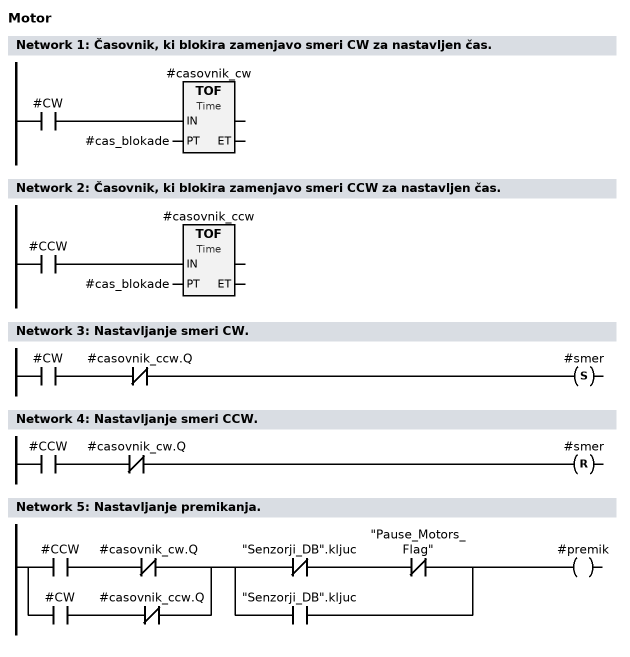
   #casovnik_cw.TOF(IN := #CW, PT := #cas_blokade);
END_REGION

REGION Network 2: Časovnik, ki blokira zamenjavo smeri CCW za nastavljen čas.
   #casovnik_ccw.TOF(IN := #CCW, PT := #cas_blokade);
END_REGION

REGION Network 3: Nastavljanje smeri CW.
   RUNG wire#powerrail
      Contact( #CW )
      I_Contact( #casovnik_ccw.Q )
      S_Coil( #smer )
   END_RUNG
   // the same network as SCL:
   IF #CW AND NOT #casovnik_ccw.Q THEN #smer := TRUE; END_IF;
END_REGION

REGION Network 4: Nastavljanje smeri CCW.
   RUNG wire#powerrail
      Contact( #CCW )
      I_Contact( #casovnik_cw.Q )
      R_Coil( #smer )
   END_RUNG
   // the same network as SCL:
   IF #CCW AND NOT #casovnik_cw.Q THEN #smer := FALSE; END_IF;
END_REGION

REGION Network 5: Nastavljanje premikanja.
   RUNG wire#powerrail
      Contact( #CCW )
      I_Contact( #casovnik_cw.Q )
      wire#w1
      I_Contact( "Senzorji_DB".kljuc )
      I_Contact( "Pause_Motors_Flag" )
      wire#w2
      Coil( #premik )
   END_RUNG
   RUNG wire#powerrail
      Contact( #CW )
      I_Contact( #casovnik_ccw.Q )
   END_RUNG wire#w1
   RUNG wire#w1
      Contact( "Senzorji_DB".kljuc )
   END_RUNG wire#w2
   // the same network as SCL:
   #premik := ((#CCW AND NOT #casovnik_cw.Q) OR (#CW AND NOT #casovnik_ccw.Q)) AND ((NOT "Senzorji_DB".kljuc AND NOT "Pause_Motors_Flag") OR "Senzorji_DB".kljuc);
END_REGION
END_FUNCTION_BLOCK

FUNCTION_BLOCK "Motorji"   // FB3, LAD
TITLE = Nastavljanje vseh različnih motorjev.
{ S7_Optimized_Access := 'FALSE' }
VERSION : 0.1
BEGIN

REGION Network 1: Izbira motorja
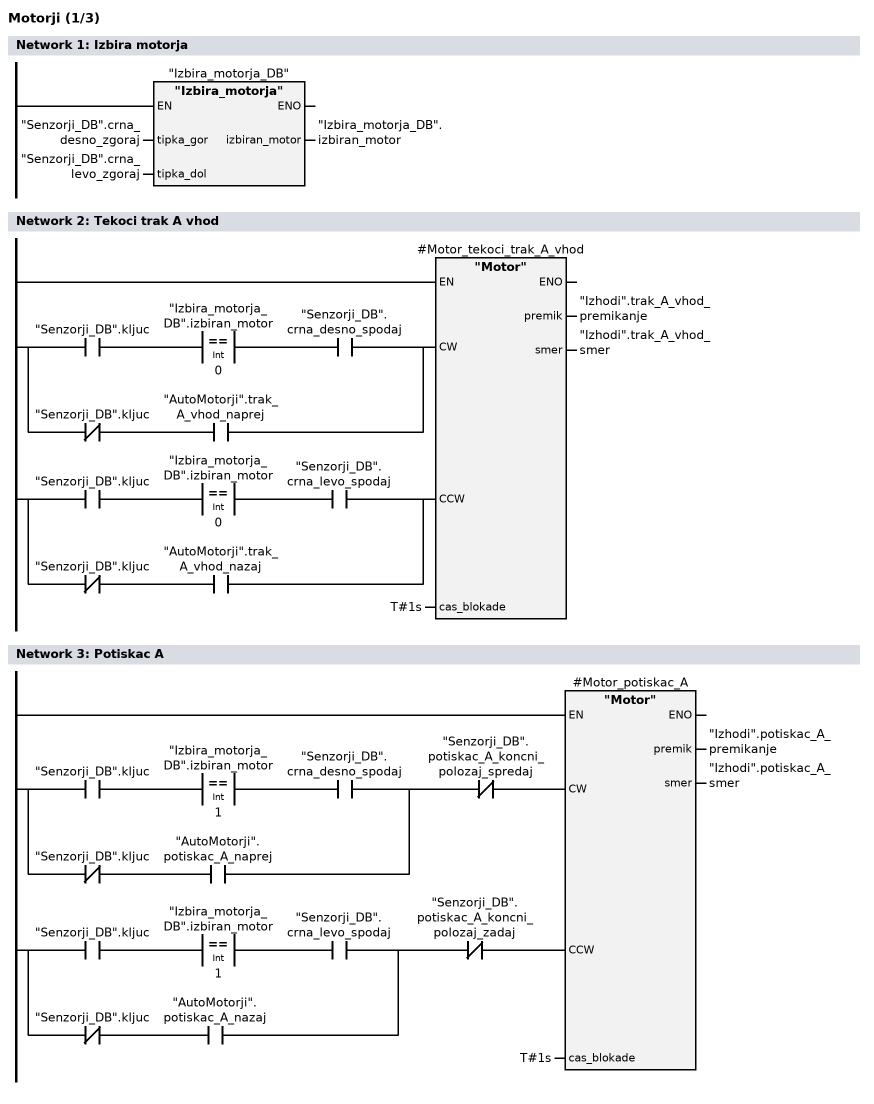
   RUNG wire#powerrail
      "Izbira_motorja_DB"(tipka_gor := "Senzorji_DB".crna_desno_zgoraj, tipka_dol := "Senzorji_DB".crna_levo_zgoraj, izbiran_motor => "Izbira_motorja_DB".izbiran_motor)
   END_RUNG
   // the same network as SCL:
   "Izbira_motorja_DB"(tipka_gor := "Senzorji_DB".crna_desno_zgoraj,   // "Izbira_motorja"
                       tipka_dol := "Senzorji_DB".crna_levo_zgoraj,
                       izbiran_motor => "Izbira_motorja_DB".izbiran_motor);
END_REGION

REGION Network 2: Tekoci trak A vhod
   RUNG wire#powerrail
      #Motor_tekoci_trak_A_vhod(CW := wire#w1, CCW := wire#w2, cas_blokade := T#1s, premik => "Izhodi".trak_A_vhod_premikanje, smer => "Izhodi".trak_A_vhod_smer)
   END_RUNG
   RUNG wire#powerrail
      Contact( "Senzorji_DB".kljuc )
      { S7_Templates := "SrcType := Int" } EQ_Contact(in1 := "Izbira_motorja_DB".izbiran_motor, in2 := 0)
      Contact( "Senzorji_DB".crna_desno_spodaj )
   END_RUNG wire#w1
   RUNG wire#powerrail
      I_Contact( "Senzorji_DB".kljuc )
      Contact( "AutoMotorji".trak_A_vhod_naprej )
   END_RUNG wire#w1
   RUNG wire#powerrail
      Contact( "Senzorji_DB".kljuc )
      { S7_Templates := "SrcType := Int" } EQ_Contact(in1 := "Izbira_motorja_DB".izbiran_motor, in2 := 0)
      Contact( "Senzorji_DB".crna_levo_spodaj )
   END_RUNG wire#w2
   RUNG wire#powerrail
      I_Contact( "Senzorji_DB".kljuc )
      Contact( "AutoMotorji".trak_A_vhod_nazaj )
   END_RUNG wire#w2
   // the same network as SCL:
   #Motor_tekoci_trak_A_vhod(CW := ("Senzorji_DB".kljuc AND ("Izbira_motorja_DB".izbiran_motor = 0) AND "Senzorji_DB".crna_desno_spodaj) OR (NOT "Senzorji_DB".kljuc AND "AutoMotorji".trak_A_vhod_naprej),   // "Motor"
                           CCW := ("Senzorji_DB".kljuc AND ("Izbira_motorja_DB".izbiran_motor = 0) AND "Senzorji_DB".crna_levo_spodaj) OR (NOT "Senzorji_DB".kljuc AND "AutoMotorji".trak_A_vhod_nazaj),
                           cas_blokade := T#1s,
                           premik => "Izhodi".trak_A_vhod_premikanje,
                           smer => "Izhodi".trak_A_vhod_smer);
END_REGION

REGION Network 3: Potiskac A
   RUNG wire#powerrail
      #Motor_potiskac_A(CW := wire#w2, CCW := wire#w4, cas_blokade := T#1s, premik => "Izhodi".potiskac_A_premikanje, smer => "Izhodi".potiskac_A_smer)
   END_RUNG
   RUNG wire#powerrail
      Contact( "Senzorji_DB".kljuc )
      { S7_Templates := "SrcType := Int" } EQ_Contact(in1 := "Izbira_motorja_DB".izbiran_motor, in2 := 1)
      Contact( "Senzorji_DB".crna_desno_spodaj )
      wire#w1
      I_Contact( "Senzorji_DB".potiskac_A_koncni_polozaj_spredaj )
   END_RUNG wire#w2
   RUNG wire#powerrail
      I_Contact( "Senzorji_DB".kljuc )
      Contact( "AutoMotorji".potiskac_A_naprej )
   END_RUNG wire#w1
   RUNG wire#powerrail
      Contact( "Senzorji_DB".kljuc )
      { S7_Templates := "SrcType := Int" } EQ_Contact(in1 := "Izbira_motorja_DB".izbiran_motor, in2 := 1)
      Contact( "Senzorji_DB".crna_levo_spodaj )
      wire#w3
      I_Contact( "Senzorji_DB".potiskac_A_koncni_polozaj_zadaj )
   END_RUNG wire#w4
   RUNG wire#powerrail
      I_Contact( "Senzorji_DB".kljuc )
      Contact( "AutoMotorji".potiskac_A_nazaj )
   END_RUNG wire#w3
   // the same network as SCL:
   #Motor_potiskac_A(CW := (("Senzorji_DB".kljuc AND ("Izbira_motorja_DB".izbiran_motor = 1) AND "Senzorji_DB".crna_desno_spodaj) OR (NOT "Senzorji_DB".kljuc AND "AutoMotorji".potiskac_A_naprej)) AND NOT "Senzorji_DB".potiskac_A_koncni_polozaj_spredaj,   // "Motor"
                     CCW := (("Senzorji_DB".kljuc AND ("Izbira_motorja_DB".izbiran_motor = 1) AND "Senzorji_DB".crna_levo_spodaj) OR (NOT "Senzorji_DB".kljuc AND "AutoMotorji".potiskac_A_nazaj)) AND NOT "Senzorji_DB".potiskac_A_koncni_polozaj_zadaj,
                     cas_blokade := T#1s,
                     premik => "Izhodi".potiskac_A_premikanje,
                     smer => "Izhodi".potiskac_A_smer);
END_REGION

REGION Network 4: Tekoci trak A stroj
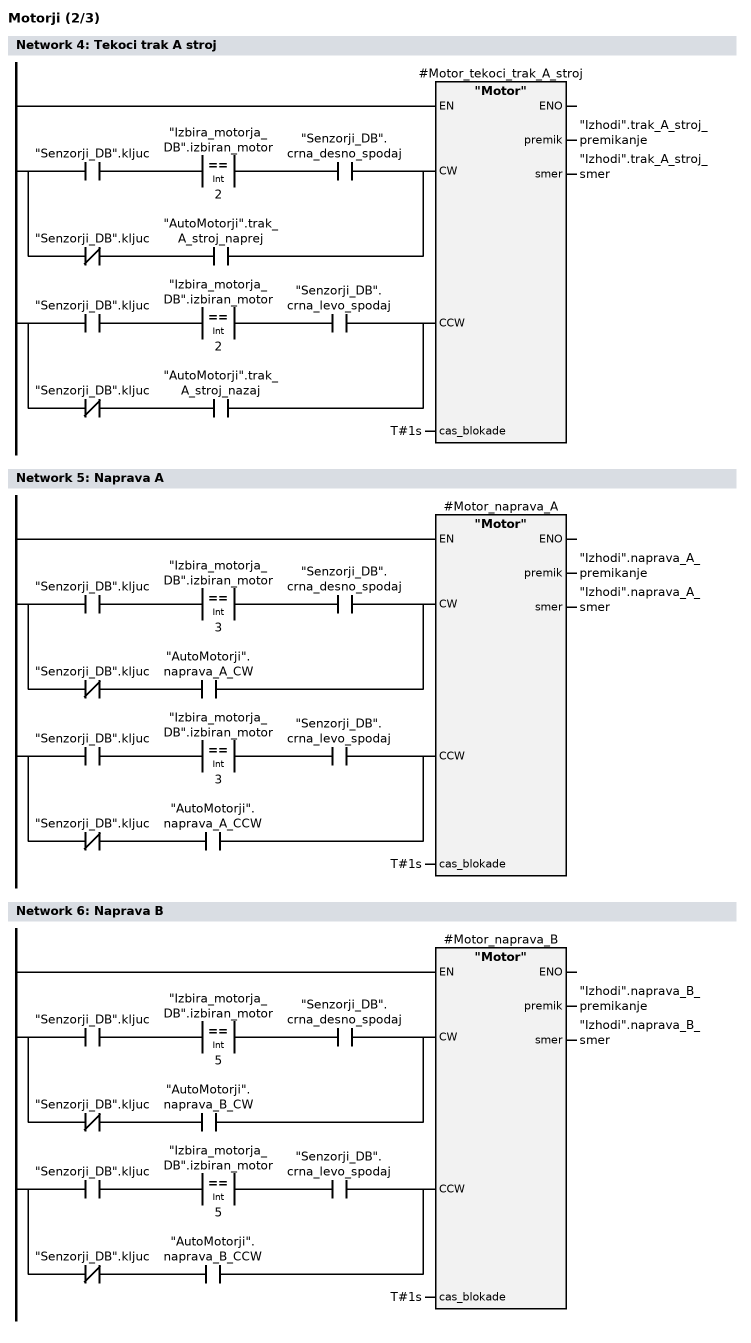
   RUNG wire#powerrail
      #Motor_tekoci_trak_A_stroj(CW := wire#w1, CCW := wire#w2, cas_blokade := T#1s, premik => "Izhodi".trak_A_stroj_premikanje, smer => "Izhodi".trak_A_stroj_smer)
   END_RUNG
   RUNG wire#powerrail
      Contact( "Senzorji_DB".kljuc )
      { S7_Templates := "SrcType := Int" } EQ_Contact(in1 := "Izbira_motorja_DB".izbiran_motor, in2 := 2)
      Contact( "Senzorji_DB".crna_desno_spodaj )
   END_RUNG wire#w1
   RUNG wire#powerrail
      I_Contact( "Senzorji_DB".kljuc )
      Contact( "AutoMotorji".trak_A_stroj_naprej )
   END_RUNG wire#w1
   RUNG wire#powerrail
      Contact( "Senzorji_DB".kljuc )
      { S7_Templates := "SrcType := Int" } EQ_Contact(in1 := "Izbira_motorja_DB".izbiran_motor, in2 := 2)
      Contact( "Senzorji_DB".crna_levo_spodaj )
   END_RUNG wire#w2
   RUNG wire#powerrail
      I_Contact( "Senzorji_DB".kljuc )
      Contact( "AutoMotorji".trak_A_stroj_nazaj )
   END_RUNG wire#w2
   // the same network as SCL:
   #Motor_tekoci_trak_A_stroj(CW := ("Senzorji_DB".kljuc AND ("Izbira_motorja_DB".izbiran_motor = 2) AND "Senzorji_DB".crna_desno_spodaj) OR (NOT "Senzorji_DB".kljuc AND "AutoMotorji".trak_A_stroj_naprej),   // "Motor"
                           CCW := ("Senzorji_DB".kljuc AND ("Izbira_motorja_DB".izbiran_motor = 2) AND "Senzorji_DB".crna_levo_spodaj) OR (NOT "Senzorji_DB".kljuc AND "AutoMotorji".trak_A_stroj_nazaj),
                           cas_blokade := T#1s,
                           premik => "Izhodi".trak_A_stroj_premikanje,
                           smer => "Izhodi".trak_A_stroj_smer);
END_REGION

REGION Network 5: Naprava A
   RUNG wire#powerrail
      #Motor_naprava_A(CW := wire#w1, CCW := wire#w2, cas_blokade := T#1s, premik => "Izhodi".naprava_A_premikanje, smer => "Izhodi".naprava_A_smer)
   END_RUNG
   RUNG wire#powerrail
      Contact( "Senzorji_DB".kljuc )
      { S7_Templates := "SrcType := Int" } EQ_Contact(in1 := "Izbira_motorja_DB".izbiran_motor, in2 := 3)
      Contact( "Senzorji_DB".crna_desno_spodaj )
   END_RUNG wire#w1
   RUNG wire#powerrail
      I_Contact( "Senzorji_DB".kljuc )
      Contact( "AutoMotorji".naprava_A_CW )
   END_RUNG wire#w1
   RUNG wire#powerrail
      Contact( "Senzorji_DB".kljuc )
      { S7_Templates := "SrcType := Int" } EQ_Contact(in1 := "Izbira_motorja_DB".izbiran_motor, in2 := 3)
      Contact( "Senzorji_DB".crna_levo_spodaj )
   END_RUNG wire#w2
   RUNG wire#powerrail
      I_Contact( "Senzorji_DB".kljuc )
      Contact( "AutoMotorji".naprava_A_CCW )
   END_RUNG wire#w2
   // the same network as SCL:
   #Motor_naprava_A(CW := ("Senzorji_DB".kljuc AND ("Izbira_motorja_DB".izbiran_motor = 3) AND "Senzorji_DB".crna_desno_spodaj) OR (NOT "Senzorji_DB".kljuc AND "AutoMotorji".naprava_A_CW),   // "Motor"
                    CCW := ("Senzorji_DB".kljuc AND ("Izbira_motorja_DB".izbiran_motor = 3) AND "Senzorji_DB".crna_levo_spodaj) OR (NOT "Senzorji_DB".kljuc AND "AutoMotorji".naprava_A_CCW),
                    cas_blokade := T#1s,
                    premik => "Izhodi".naprava_A_premikanje,
                    smer => "Izhodi".naprava_A_smer);
END_REGION

REGION Network 6: Naprava B
   RUNG wire#powerrail
      #Motor_naprava_B(CW := wire#w1, CCW := wire#w2, cas_blokade := T#1s, premik => "Izhodi".naprava_B_premikanje, smer => "Izhodi".naprava_B_smer)
   END_RUNG
   RUNG wire#powerrail
      Contact( "Senzorji_DB".kljuc )
      { S7_Templates := "SrcType := Int" } EQ_Contact(in1 := "Izbira_motorja_DB".izbiran_motor, in2 := 5)
      Contact( "Senzorji_DB".crna_desno_spodaj )
   END_RUNG wire#w1
   RUNG wire#powerrail
      I_Contact( "Senzorji_DB".kljuc )
      Contact( "AutoMotorji".naprava_B_CW )
   END_RUNG wire#w1
   RUNG wire#powerrail
      Contact( "Senzorji_DB".kljuc )
      { S7_Templates := "SrcType := Int" } EQ_Contact(in1 := "Izbira_motorja_DB".izbiran_motor, in2 := 5)
      Contact( "Senzorji_DB".crna_levo_spodaj )
   END_RUNG wire#w2
   RUNG wire#powerrail
      I_Contact( "Senzorji_DB".kljuc )
      Contact( "AutoMotorji".naprava_B_CCW )
   END_RUNG wire#w2
   // the same network as SCL:
   #Motor_naprava_B(CW := ("Senzorji_DB".kljuc AND ("Izbira_motorja_DB".izbiran_motor = 5) AND "Senzorji_DB".crna_desno_spodaj) OR (NOT "Senzorji_DB".kljuc AND "AutoMotorji".naprava_B_CW),   // "Motor"
                    CCW := ("Senzorji_DB".kljuc AND ("Izbira_motorja_DB".izbiran_motor = 5) AND "Senzorji_DB".crna_levo_spodaj) OR (NOT "Senzorji_DB".kljuc AND "AutoMotorji".naprava_B_CCW),
                    cas_blokade := T#1s,
                    premik => "Izhodi".naprava_B_premikanje,
                    smer => "Izhodi".naprava_B_smer);
END_REGION

REGION Network 7: Tekoci trak B stroj
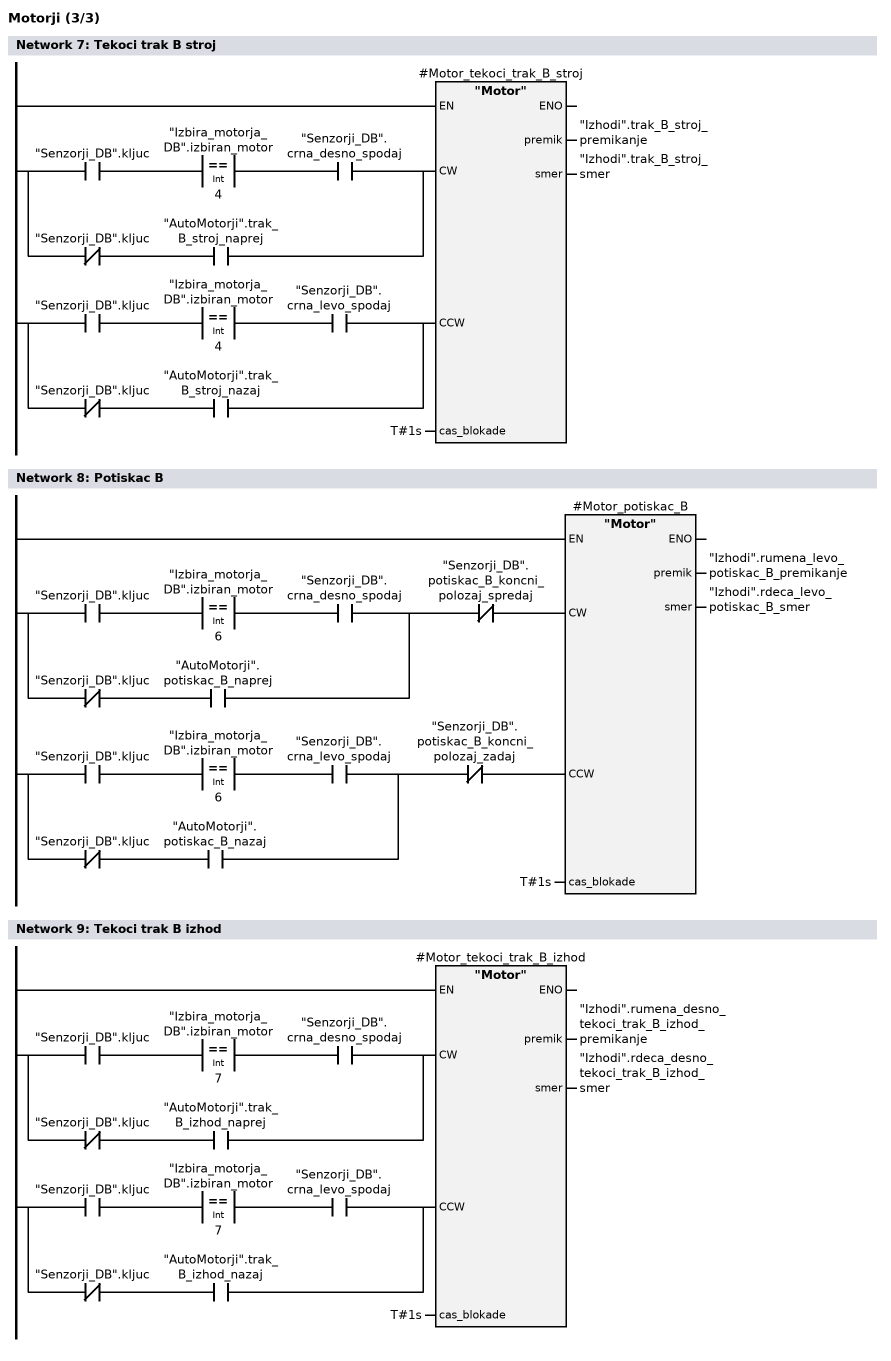
   RUNG wire#powerrail
      #Motor_tekoci_trak_B_stroj(CW := wire#w1, CCW := wire#w2, cas_blokade := T#1s, premik => "Izhodi".trak_B_stroj_premikanje, smer => "Izhodi".trak_B_stroj_smer)
   END_RUNG
   RUNG wire#powerrail
      Contact( "Senzorji_DB".kljuc )
      { S7_Templates := "SrcType := Int" } EQ_Contact(in1 := "Izbira_motorja_DB".izbiran_motor, in2 := 4)
      Contact( "Senzorji_DB".crna_desno_spodaj )
   END_RUNG wire#w1
   RUNG wire#powerrail
      I_Contact( "Senzorji_DB".kljuc )
      Contact( "AutoMotorji".trak_B_stroj_naprej )
   END_RUNG wire#w1
   RUNG wire#powerrail
      Contact( "Senzorji_DB".kljuc )
      { S7_Templates := "SrcType := Int" } EQ_Contact(in1 := "Izbira_motorja_DB".izbiran_motor, in2 := 4)
      Contact( "Senzorji_DB".crna_levo_spodaj )
   END_RUNG wire#w2
   RUNG wire#powerrail
      I_Contact( "Senzorji_DB".kljuc )
      Contact( "AutoMotorji".trak_B_stroj_nazaj )
   END_RUNG wire#w2
   // the same network as SCL:
   #Motor_tekoci_trak_B_stroj(CW := ("Senzorji_DB".kljuc AND ("Izbira_motorja_DB".izbiran_motor = 4) AND "Senzorji_DB".crna_desno_spodaj) OR (NOT "Senzorji_DB".kljuc AND "AutoMotorji".trak_B_stroj_naprej),   // "Motor"
                           CCW := ("Senzorji_DB".kljuc AND ("Izbira_motorja_DB".izbiran_motor = 4) AND "Senzorji_DB".crna_levo_spodaj) OR (NOT "Senzorji_DB".kljuc AND "AutoMotorji".trak_B_stroj_nazaj),
                           cas_blokade := T#1s,
                           premik => "Izhodi".trak_B_stroj_premikanje,
                           smer => "Izhodi".trak_B_stroj_smer);
END_REGION

REGION Network 8: Potiskac B
   RUNG wire#powerrail
      #Motor_potiskac_B(CW := wire#w2, CCW := wire#w4, cas_blokade := T#1s, premik => "Izhodi".rumena_levo_potiskac_B_premikanje, smer => "Izhodi".rdeca_levo_potiskac_B_smer)
   END_RUNG
   RUNG wire#powerrail
      Contact( "Senzorji_DB".kljuc )
      { S7_Templates := "SrcType := Int" } EQ_Contact(in1 := "Izbira_motorja_DB".izbiran_motor, in2 := 6)
      Contact( "Senzorji_DB".crna_desno_spodaj )
      wire#w1
      I_Contact( "Senzorji_DB".potiskac_B_koncni_polozaj_spredaj )
   END_RUNG wire#w2
   RUNG wire#powerrail
      I_Contact( "Senzorji_DB".kljuc )
      Contact( "AutoMotorji".potiskac_B_naprej )
   END_RUNG wire#w1
   RUNG wire#powerrail
      Contact( "Senzorji_DB".kljuc )
      { S7_Templates := "SrcType := Int" } EQ_Contact(in1 := "Izbira_motorja_DB".izbiran_motor, in2 := 6)
      Contact( "Senzorji_DB".crna_levo_spodaj )
      wire#w3
      I_Contact( "Senzorji_DB".potiskac_B_koncni_polozaj_zadaj )
   END_RUNG wire#w4
   RUNG wire#powerrail
      I_Contact( "Senzorji_DB".kljuc )
      Contact( "AutoMotorji".potiskac_B_nazaj )
   END_RUNG wire#w3
   // the same network as SCL:
   #Motor_potiskac_B(CW := (("Senzorji_DB".kljuc AND ("Izbira_motorja_DB".izbiran_motor = 6) AND "Senzorji_DB".crna_desno_spodaj) OR (NOT "Senzorji_DB".kljuc AND "AutoMotorji".potiskac_B_naprej)) AND NOT "Senzorji_DB".potiskac_B_koncni_polozaj_spredaj,   // "Motor"
                     CCW := (("Senzorji_DB".kljuc AND ("Izbira_motorja_DB".izbiran_motor = 6) AND "Senzorji_DB".crna_levo_spodaj) OR (NOT "Senzorji_DB".kljuc AND "AutoMotorji".potiskac_B_nazaj)) AND NOT "Senzorji_DB".potiskac_B_koncni_polozaj_zadaj,
                     cas_blokade := T#1s,
                     premik => "Izhodi".rumena_levo_potiskac_B_premikanje,
                     smer => "Izhodi".rdeca_levo_potiskac_B_smer);
END_REGION

REGION Network 9: Tekoci trak B izhod
   RUNG wire#powerrail
      #Motor_tekoci_trak_B_izhod(CW := wire#w1, CCW := wire#w2, cas_blokade := T#1s, premik => "Izhodi".rumena_desno_tekoci_trak_B_izhod_premikanje, smer => "Izhodi".rdeca_desno_tekoci_trak_B_izhod_smer)
   END_RUNG
   RUNG wire#powerrail
      Contact( "Senzorji_DB".kljuc )
      { S7_Templates := "SrcType := Int" } EQ_Contact(in1 := "Izbira_motorja_DB".izbiran_motor, in2 := 7)
      Contact( "Senzorji_DB".crna_desno_spodaj )
   END_RUNG wire#w1
   RUNG wire#powerrail
      I_Contact( "Senzorji_DB".kljuc )
      Contact( "AutoMotorji".trak_B_izhod_naprej )
   END_RUNG wire#w1
   RUNG wire#powerrail
      Contact( "Senzorji_DB".kljuc )
      { S7_Templates := "SrcType := Int" } EQ_Contact(in1 := "Izbira_motorja_DB".izbiran_motor, in2 := 7)
      Contact( "Senzorji_DB".crna_levo_spodaj )
   END_RUNG wire#w2
   RUNG wire#powerrail
      I_Contact( "Senzorji_DB".kljuc )
      Contact( "AutoMotorji".trak_B_izhod_nazaj )
   END_RUNG wire#w2
   // the same network as SCL:
   #Motor_tekoci_trak_B_izhod(CW := ("Senzorji_DB".kljuc AND ("Izbira_motorja_DB".izbiran_motor = 7) AND "Senzorji_DB".crna_desno_spodaj) OR (NOT "Senzorji_DB".kljuc AND "AutoMotorji".trak_B_izhod_naprej),   // "Motor"
                           CCW := ("Senzorji_DB".kljuc AND ("Izbira_motorja_DB".izbiran_motor = 7) AND "Senzorji_DB".crna_levo_spodaj) OR (NOT "Senzorji_DB".kljuc AND "AutoMotorji".trak_B_izhod_nazaj),
                           cas_blokade := T#1s,
                           premik => "Izhodi".rumena_desno_tekoci_trak_B_izhod_premikanje,
                           smer => "Izhodi".rdeca_desno_tekoci_trak_B_izhod_smer);
END_REGION
END_FUNCTION_BLOCK

(* ===== HMI "HMI_RT_1" =====
connection "HMI_Connection_1": ETHERNET, SIMATIC S7 300/400 MPI

HMI tags "Default tag table"
   "SCADA_alarm_aktive_globalno" : Bool, 100 ms
   "SCADA_alarm_potrditev" : Bool, 100 ms
   "SCADA_alarmi" : Word, 100 ms
   "SCADA_recept_vrtanje1" : Bool, 100 ms
   "SCADA_recept_cas_vrtanja1" : Time, 100 ms
   "SCADA_recept_vrtanje2" : Bool, 100 ms
   "SCADA_recept_cas_vrtanja2" : Time, 100 ms
   "SCADA_recept_smer_1" : Bool, 100 ms
   "SCADA_recept_smer_2" : Bool, 100 ms
   "Lokacije_DB_L1_vhod_1_zasedenost" : Bool, 100 ms
   "L1_L2_CNT_CV" : Int, 100 ms
   "Lokacije_DB_L2_vhod_2_zasedenost" : Bool, 100 ms
   "L2_L3_CNT_CV" : Int, 100 ms
   "Lokacije_DB_L3_potiskac_A_zasedenost" : Bool, 100 ms
   "L3_L4_CNT_CV" : Int, 100 ms
   "Lokacije_DB_L4_naprava_A_zasedenost" : Bool, 100 ms
   "Lokacije_DB_L5_naprava_B_zasedenost" : Bool, 100 ms
   "Lokacije_DB_L6_potiskac_B_zasedenost" : Bool, 100 ms
   "Lokacije_DB_L7_izhod_zasedenost" : Bool, 100 ms
   "SCADAVisual_DB_l3_l4_visibily" : Bool, 100 ms
   "L4_L5_CNT_CV" : Int, 100 ms
   "L5_L6_CNT_CV" : Int, 100 ms
   "L6_L7_CNT_CV" : Int, 100 ms
   "SCADAVisual_DB_l6_l7_visibily" : Bool, 100 ms
   "Senzorji_DB_fotocelica_material_na_vhodu" : Bool, 100 ms
   "Senzorji_DB_fotocelica_materal_pred_potiskacem" : Bool, 100 ms
   "Senzorji_DB_fotocelica_material_pod_napravo_A" : Bool, 100 ms
   "Senzorji_DB_fotocelica_material_pod_napravo_B" : Bool, 100 ms
   "Senzorji_DB_fotocelica_material_na_izhodu" : Bool, 100 ms
   "Senzorji_DB_potiskac_A_koncni_polozaj_zadaj" : Bool, 100 ms
   "Senzorji_DB_potiskac_A_koncni_polozaj_spredaj" : Bool, 100 ms
   "SCADAVisual_DB_potiskac_A_levo" : Bool, 100 ms
   "SCADAVisual_DB_potiskac_A_desno" : Bool, 100 ms
   "SCADAVisual_DB;potiskac_B_dol" : Bool, 100 ms
   "SCADAVisual_DB;potiskac_B_gor" : Bool, 100 ms
   "Senzorji_DB;potiskac_B_koncni_polozaj_zadaj" : Bool, 100 ms
   "Senzorji_DB;potiskac_B_koncni_polozaj_spredaj" : Bool, 100 ms
   "SCADAVisual_DB;trak_vhod_nazaj" : Bool, 100 ms
   "SCADAVisual_DB;trak_vhod_naprej" : Bool, 100 ms
   "SCADAVisual_DB;trak_A_naprej" : Bool, 100 ms
   "SCADAVisual_DB;trak_A_nazaj" : Bool, 100 ms
   "SCADAVisual_DB;trak_B_nazaj" : Bool, 100 ms
   "SCADAVisual_DB;trak_izhod_naprej" : Bool, 100 ms
   "SCADAVisual_DB;trak_izhod_nazaj" : Bool, 100 ms
   "SCADAVisual_DB;trak_B_naprej" : Bool, 100 ms
   "SCADAVisual_DB;l3_visibility" : Bool, 100 ms
   "SCADAVisual_DB;l6_visibility" : Bool, 100 ms
   "Auto_2_A_Naprava_DB;casVrtanja" : DInt, 100 ms
   "Auto_2_A_Naprava_DB;maxCasVrtanja" : DInt, 100 ms
   "Auto_3_B_Naprava_DB;casVrtanja" : DInt, 100 ms
   "Auto_3_B_Naprava_DB;maxCasVrtanja" : DInt, 100 ms
   "Lokacije_DB;L1_vhod_1;ID" : Int, 100 ms
   "Lokacije_DB;L2_vhod_2;ID" : Int, 100 ms
   "Lokacije_DB;L3_potiskac_A;ID" : Int, 100 ms
   "Lokacije_DB;L4_naprava_A;ID" : Int, 100 ms
   "Lokacije_DB;L5_naprava_B;ID" : Int, 100 ms
   "Lokacije_DB;L6_potiskac_B;ID" : Int, 100 ms
   "Lokacije_DB;L7_izhod;ID" : Int, 100 ms
   "Lokacije_DB;L4_naprava_A;recept;smer_1" : Bool, 100 ms
   "Lokacije_DB;L5_naprava_B;recept;smer_2" : Bool, 100 ms
   "SCADA;recept_num" : Int, 100 ms
   "Lokacije_DB;L1_vhod_1;recept;ID_recepta" : Int, 100 ms
   "Lokacije_DB;L6_potiskac_B;recept;ID_recepta" : Int, 100 ms
   "SCADAVisual_DB;naprava_A_leva" : Bool, 100 ms
   "SCADAVisual_DB;naprava_A_desna" : Bool, 100 ms
   "SCADAVisual_DB;naprava_B_leva" : Bool, 100 ms
   "SCADAVisual_DB;naprava_B_desna" : Bool, 100 ms
   "Lokacije_DB;L2_vhod_2;recept;ID_recepta" : Int, 100 ms
   "Lokacije_DB;L3_potiskac_A;recept;ID_recepta" : Int, 100 ms
   "Lokacije_DB;L4_naprava_A;recept;ID_recepta" : Int, 100 ms
   "Lokacije_DB;L5_naprava_B;recept;ID_recepta" : Int, 100 ms
   "Lokacije_DB;L7_izhod;recept;ID_recepta" : Int, 100 ms
   "SCADA;alarmi{0}" : Bool, 1 s
   "SCADA;alarmi{1}" : Bool, 1 s
   "SCADA;alarmi{2}" : Bool, 1 s
   "SCADA;alarmi{3}" : Bool, 1 s
   "SCADA;alarmi{4}" : Bool, 1 s
   "SCADA;alarmi{5}" : Bool, 1 s
   "SCADA;alarmi{6}" : Bool, 1 s
   "SCADA;alarmi{7}" : Bool, 1 s
   "SCADA;alarmi{8}" : Bool, 1 s
   "SCADA;alarmi{9}" : Bool, 1 s
   "SCADA;alarmi{10}" : Bool, 1 s
   "SCADA;alarmi{11}" : Bool, 1 s
   "SCADA;alarmi{12}" : Bool, 1 s
   "SCADA;alarmi{13}" : Bool, 1 s
   "SCADA;alarmi{14}" : Bool, 1 s
   "SCADA;alarmi{15}" : Bool, 1 s

discrete alarms
   1: '', class Info, trigger "SCADA_alarmi" bit 0
   2: '', class Warnings, trigger "SCADA_alarmi" bit 1
   3: '', class Info, trigger "SCADA_alarmi" bit 2
   4: '', class Info, trigger "SCADA_alarmi" bit 3
   5: '', class Errors, trigger "SCADA_alarmi" bit 4
   6: '', class Errors, trigger "SCADA_alarmi" bit 5
   7: '', class Errors, trigger "SCADA_alarmi" bit 6
   8: '', class Warnings, trigger "SCADA_alarmi" bit 7
   9: '', class Errors, trigger "SCADA_alarmi" bit 8
   10: '', class Errors, trigger "SCADA_alarmi" bit 9
   11: '', class Errors, trigger "SCADA_alarmi" bit 10
   12: '', class Errors, trigger "SCADA_alarmi" bit 11
   13: '', class Errors, trigger "SCADA_alarmi" bit 12
   14: '', class Errors, trigger "SCADA_alarmi" bit 13
   15: '', class Errors, trigger "SCADA_alarmi" bit 14
   16: '', class Errors, trigger "SCADA_alarmi" bit 15

recipe "Marmor": vrtanje1 <- "SCADA_recept_vrtanje1", cas_vrtanja1 <- "SCADA_recept_cas_vrtanja1", vrtanje2 <- "SCADA_recept_vrtanje2", cas_vrtanja2 <- "SCADA_recept_cas_vrtanja2", smer_1 <- "SCADA_recept_smer_1", smer_2 <- "SCADA_recept_smer_2"

screen "main" 1024x768, template "Predloga"
   GraphicView "Graphic view_1" at 946,18 size 50x32
   Bar "Bar_1" at 344,173 size 111x34
   Bar "Bar_2" at 525,173 size 111x34
   TextField "Text field_2" at 130,509 size 35x20
   TextField "Text field_3" at 307,422 size 75x20
   IOField "I/O field_1" at 166,508 size 20x20
   IOField "I/O field_2" at 382,423 size 20x20
   IOField "I/O field_3" at 165,312 size 20x20
   IOField "I/O field_5" at 165,230 size 20x20
   IOField "I/O field_7" at 379,150 size 20x20
   IOField "I/O field_9" at 560,150 size 20x20
   IOField "I/O field_11" at 793,510 size 20x20
   IOField "I/O field_13" at 793,230 size 20x20
   TextField "Text field_1" at 307,451 size 75x14
   TextField "Text field_4" at 307,471 size 75x14
   TextField "Text field_5" at 307,491 size 54x14
   TextField "Text field_6" at 307,511 size 54x14
   TextField "Text field_7" at 307,531 size 47x14
   TextField "Text field_8" at 307,551 size 47x14
   IOField "I/O field_4" at 382,450 size 14x15
   IOField "I/O field_6" at 382,470 size 14x15
   IOField "I/O field_8" at 382,490 size 14x15
   IOField "I/O field_10" at 382,510 size 14x15
   IOField "I/O field_12" at 382,530 size 42x15
   IOField "I/O field_14" at 382,550 size 42x15
   IOField "I/O field_15" at 166,530 size 20x20
   IOField "I/O field_16" at 793,252 size 20x20
   TextField "Text field_9" at 90,528 size 75x20
   IOField "I/O field_17" at 165,334 size 20x20
   IOField "I/O field_18" at 165,252 size 20x20
   IOField "I/O field_19" at 401,150 size 20x20
   IOField "I/O field_20" at 582,150 size 20x20
   IOField "I/O field_21" at 793,532 size 20x20
   TextField "Text field_10" at 923,4 size 71x14
   TextField "Text field_11" at 936,49 size 65x14
   TextField "Text field_12" at 992,4 size 22x14

screen "Alarmi" 1024x768, template "Predloga"
   AlarmView "Alarm view_1" at 108,110 size 810x383
   Button "Button_1" at 108,515 size 810x51
   TextField "Text field_1" at 469,30 size 88x34

Template "Predloga" 1024x768
   Button "Template_Button_1" at 108,645 size 214x68
   Button "Template_Button_2" at 405,646 size 214x68
   Button "Template_Button_3" at 702,645 size 214x68

screen "Recepti" 1024x768, template "Predloga"
   TextField "Text field_1" at 469,30 size 100x34
   RecipeView "Recipe view_1" at 173,81 size 712x427
*)